(* PLC project prj, KAIST_DSLAB noNameNow 1, author bwkim *)
(* stored: creationDateTime 2015-7-12T01:57:08, modificationDateTime 2015-7-12T01:57:08 *)

PROGRAM Program1____sub1
  VAR
    ton1 : null;
  END_VAR
  VAR_INPUT
    PV_OUT : INT;
  END_VAR
  VAR_INPUT
    TSP : INT := 26805;
  END_VAR
  VAR_INPUT
    K_DELAY : INT := 100;
  END_VAR
  VAR_OUTPUT
    TON_et : INT;
  END_VAR
  VAR_IN_OUT
    TRIP_LOGIC : BOOL := FALSE;
  END_VAR

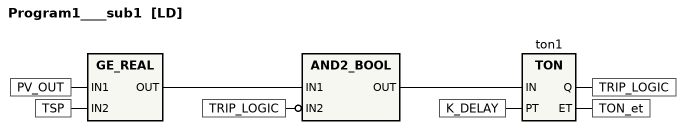
(* LD diagram, written out as Structured Text *)
ton1(IN := AND2_BOOL(GE_REAL(PV_OUT, TSP), NOT TRIP_LOGIC), PT := K_DELAY);
TRIP_LOGIC := ton1.Q;
TON_et := ton1.ET;
END_PROGRAM
